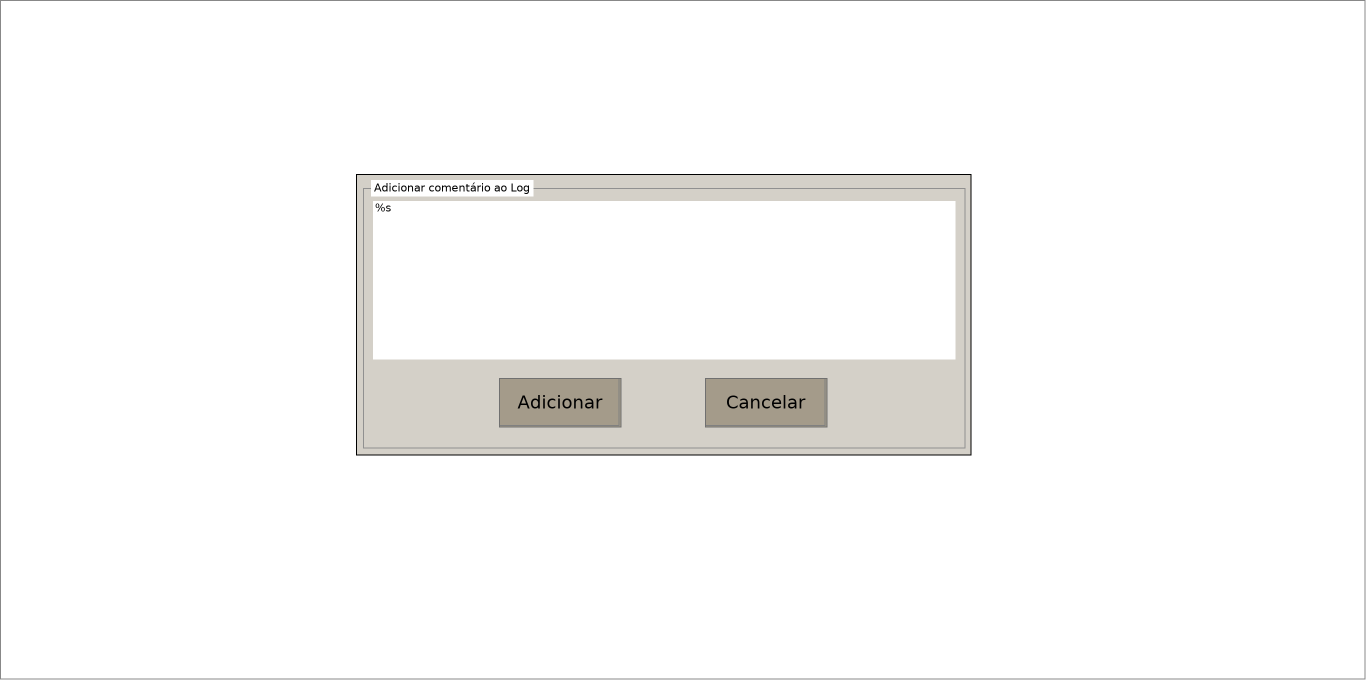
VISUALIZATION addComment  // 1366x680
    Rectangle (356,174 615x281)
    GroupBox (363,180 602x268), "Adicionar comentário ao Log"
        Textfield (9,20 584x160), "%s", text variable: GVL.addTextLog
            OnMouseDown: write GVL.addTextLog via VisuDialogs.Keypad, format ADD COMMENT
        Button (136,198 122x49), "Adicionar"
            OnMouseClick: CloseDialog Dialog=addComment, Result=OK, NumpadKeypadSet=True
            OnMouseClick: execute {
                ///// GERADOR DE LOG -------------------------------------------------------------
                gvl.logRegister19:= gvl.addTextLog;
            }
        Button (342,198 122x49), "Cancelar"
            OnMouseClick: CloseDialog Dialog=addComment, Result=OK, NumpadKeypadSet=True
END_VISUALIZATION

(* stored: Version 1.1.0.1, ProductVersion 3.1.4024.12
   Visu addComment: Id {23d1adb6-6943-40a1-a5d4-7eac95b3e61b} *)
